// Mitsubishi GX Works2 project: 22   PLC: FX3G

// task Task_01 (event TRUE, interval 0, priority 31): POU_01

PROGRAM POU_01
VAR
  gas : INT;
  ton1 : TON;
END_VAR
IF M8002 THEN
	gas := 0;
END_IF;

CASE gas OF
0:
Y0:=FALSE;
Y1:=FALSE;
Y2:=FALSE;
Y3:=FALSE;

IF M1=TRUE THEN
	gas:=1;
END_IF;

IF M2=TRUE THEN
	gas:=11;
END_IF;

IF M3=TRUE THEN
	gas:=21;
END_IF;

1:
Y0:=TRUE;
ton1(IN := NOT ton1.Q, PT := T#10s);
	IF ton1.Q THEN
		Y0:=FALSE;
		gas:=2;
	END_IF;

2:
Y1:=TRUE;
ton1(IN := NOT ton1.Q, PT := T#10s);
	IF ton1.Q THEN
		Y1:=FALSE;
		gas:=3;
	END_IF;

3:
Y2:=TRUE;
ton1(IN := NOT ton1.Q, PT := T#10s);
	IF ton1.Q THEN
		Y2:=FALSE;
		gas:=4;
	END_IF;
	
4:
Y3:=TRUE;
ton1(IN := NOT ton1.Q, PT := T#10s);
	IF ton1.Q THEN
		gas:=0;
	END_IF;

11:
Y3:=TRUE;
ton1(IN := NOT ton1.Q, PT := T#10s);
	IF ton1.Q THEN
		gas:=0;
	END_IF;

21:
Y0:=TRUE;
ton1(IN := NOT ton1.Q, PT := T#5s);
	IF ton1.Q THEN
		Y0:=FALSE;
		gas:=22;
	END_IF;

22:
Y1:=TRUE;
ton1(IN := NOT ton1.Q, PT := T#5s);
	IF ton1.Q THEN
		Y1:=FALSE;
		gas:=23;
	END_IF;

23:
Y2:=TRUE;
ton1(IN := NOT ton1.Q, PT := T#5s);
	IF ton1.Q THEN
		Y2:=FALSE;
		gas:=24;
	END_IF;
	
24:
Y3:=TRUE;
ton1(IN := NOT ton1.Q, PT := T#5s);
	IF ton1.Q THEN
		gas:=0;
	END_IF;
END_CASE;
END_PROGRAM
